# EPICS autosave request: iocBoot/ioc13ida_linux/Galil_positions.req
file "CARS_32_motor_positions.req",    P=$(P)
